PROGRAM simIniciaProg_Manual_2
VAR
	bSimIniciaProg: BOOL:= FALSE;
	posicaoAtual: STRING;
	envialog: STRING;
	bGravarConfigPosicao_Reator: BOOL;
END_VAR


gvl_p.arrStatusEstufas[gvl.actEst].startManual := TRUE;

bGravarConfigPosicao_Reator:= TRUE;

END_PROGRAM

(* stored: Version 1.1.0.1, ProductVersion 3.1.4024.12
   POU simIniciaProg_Manual_2: Id {de71e216-96e1-4ffc-9b8a-4438f85a96dc}, SpecialFunc None *)
